{attribute 'qualified_only'}
VAR_GLOBAL
	// Database record driver
	fbInfluxDBRecorder	:RecordInfluxDB(DBID := 1);
END_VAR

(* stored: Version 1.1.0.1, ProductVersion 3.1.4024.12
   GVL GVL: Id {6f3eba4c-e974-471d-8fe6-3536cf2de0a1} *)
